TYPE ST_ZAxisCommand :
STRUCT
    (* 请求使能 Z 轴。 *)
    bEnable : BOOL;
    (* 请求复位 Z 轴错误。 *)
    bReset : BOOL;
    (* 请求受控停止 Z 轴。 *)
    bStop : BOOL;
    (* 请求执行标准 NC 回零。 *)
    bHome : BOOL;
    (* 请求标准绝对定位。 *)
    bMoveAbsolute : BOOL;
    (* 请求标准速度运动。 *)
    bMoveVelocity : BOOL;
    (* 请求由外部设定值适配器接管。 *)
    bUseExternalSetpoint : BOOL;
    (* 回零完成后使用的参考位置，向下为正，单位毫米。 *)
    rHomePosition_mm : LREAL;
    (* 绝对位置目标，向下为正，单位毫米。 *)
    rPosition_mm : LREAL;
    (* 速度目标，向下为正，单位毫米每秒。 *)
    rVelocity_mm_s : LREAL;
    (* 加速度限制，单位毫米每二次方秒。 *)
    rAcceleration_mm_s2 : LREAL;
    (* 减速度限制，单位毫米每二次方秒。 *)
    rDeceleration_mm_s2 : LREAL;
    (* 请求取得控制权的命令所有者。 *)
    eOwnerRequest : E_ZCommandOwner;
END_STRUCT
END_TYPE

(* stored: Version 1.1.0.1
   DUT ST_ZAxisCommand: Id {D2000000-0000-4000-8000-000000000005} *)
